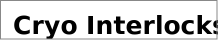
VISUALIZATION VISU_HMI_CRYO_INTERLOCKS  // 218x40
    Label (10,10 208x30), "Cryo Interlocks"
END_VISUALIZATION

(* stored: Version 1.1.0.1, ProductVersion 3.1.4024.14
   Visu VISU_HMI_CRYO_INTERLOCKS: Id {d848a9bf-8392-4f69-8cfd-372af980ba32} *)
